{attribute 'linkalways'} 
{attribute 'no_explicit_call' := 'This FB is a CLASS and must be accessed using methods or properties'}
{attribute 'enable_dynamic_creation'}
FUNCTION_BLOCK Node_F_VN_MedianElementElementwise_TcVnVector2_SINT EXTENDS VisionNode
VAR
    ipContainer : _ITcVnContainer;
    aMedian : _TcVnVector2_SINT;
    hrPrev : _HRESULT(S_OK);
    hresult : _HRESULT(S_OK);
END_VAR

METHOD PUBLIC  Clone : I_Node
VAR
	pNode : POINTER TO Node_F_VN_MedianElementElementwise_TcVnVector2_SINT;
END_VAR
pNode := __NEW(Node_F_VN_MedianElementElementwise_TcVnVector2_SINT);
Clone := pNode^;
END_METHOD

METHOD FB_init : BOOL
VAR_INPUT
	bInitRetains : BOOL; // if TRUE, the retain variables are initialized (warm start / cold start)
	bInCopyCode : BOOL;  // if TRUE, the instance afterwards gets moved into the copy code (online change)
END_VAR
AddInput('ipContainer', ipContainer);
AddInput('hrPrev', hrPrev);
AddOutput('ipContainer', ipContainer);
AddOutput('aMedian', aMedian);
AddOutput('hresult',hresult);
END_METHOD

METHOD PROTECTED OnExecute
hresult.Value := F_VN_MedianElementElementwise_TcVnVector2_SINT(
    ipContainer := ipContainer.Value,
    aMedian := aMedian.Value,
    hrPrev:= hrPrev.Value);
END_METHOD

METHOD PUBLIC PreExecutionCheck
VAR_INPUT
	Check : I_PreExecutionChecks;
END_VAR
Check.IsTrue(ipContainer.IsValid, 'ipContainer must be a valid container');
Check.IsTrue(ipContainer.IsType(TC_GLOBAL_CONST_LIST.ContainerType_Vector_TcVnVector2_SINT), 'ipContainer contains incorrect type');
END_METHOD

END_FUNCTION_BLOCK

(* stored: Version 1.1.0.1, ProductVersion 3.1.4026.13
   POU Node_F_VN_MedianElementElementwise_TcVnVector2_SINT: Id {25cb2f7f-5bfd-4962-9cd3-d12a62300861}, SpecialFunc None
   Folder Constructor: Id {916d0b59-ccc1-4d66-981a-6a6a00d5e3c1}
   Method Clone: Id {8e86bb6d-2051-4e2d-91d4-a4a1d985826e}
   Method FB_init: Id {6cb2bee7-d6f8-4cab-92bb-d288b224cf53}
   Method OnExecute: Id {24e847a3-6298-4bf9-89fc-aa7eae518423}
   Method PreExecutionCheck: Id {9a9a587f-7ca4-46a1-a232-e94eaa941b7e} *)
